{region '#Template'}
	{attribute 'Version' := '5.0.0.0'}
	{attribute 'Tags' := '"LCID": "1031", "Text": "Gebäudeautomation, Wetterdaten"'}
	{attribute 'Tags' := '"LCID": "1033", "Text": "Building automation, Weather data"'}
	{attribute 'Using' := '"Type": "Template", "URI": "BA2_Param"'}
	{attribute 'Using' := '"Type": "Template", "URI": "Site"'}		  
	{attribute 'Using' := '"Type": "Template", "URI": "ST_BA_GeneralSettings"'}
	{attribute 'Description' := '"LCID": "1031", "Text": "Gebäude Wetterdaten"'}
	{attribute 'Description' := '"LCID": "1033", "Text": "Building Weather data"'}
{endregion}
FUNCTION_BLOCK FB_BA_WeatherData EXTENDS FB_BA_View
VAR_INPUT CONSTANT
	WthParam				: FB_BA_WeatherParameter;	
END_VAR
VAR // added by the converter: edge detectors and wires of the graphical bodies
    _s1 : ST_BA_GeneralSettings;
END_VAR

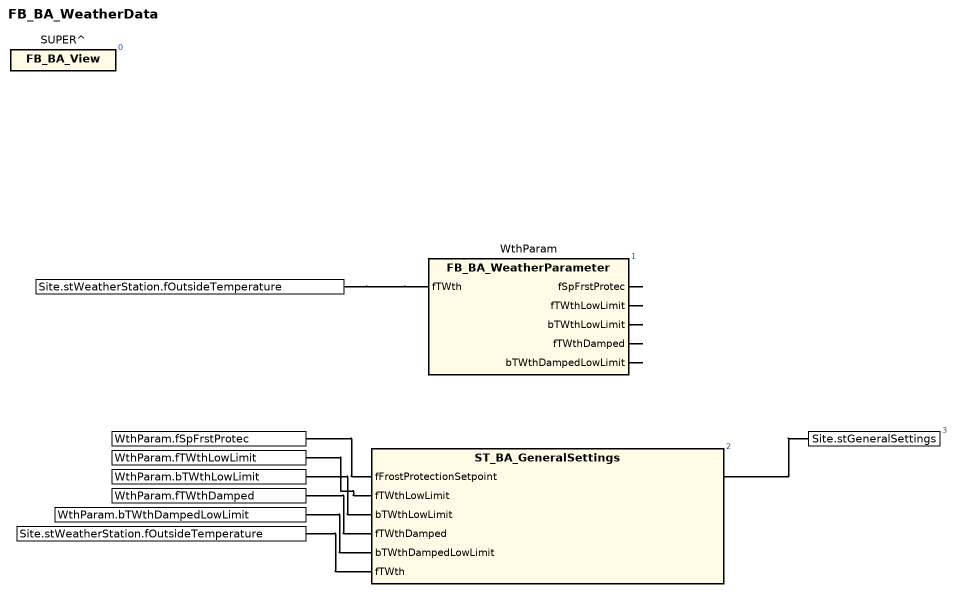
SUPER^(); // FB_BA_View
WthParam(fTWth := Site.stWeatherStation.fOutsideTemperature); // FB_BA_WeatherParameter
// compose _s1 : ST_BA_GeneralSettings
_s1.fFrostProtectionSetpoint := WthParam.fSpFrstProtec;
_s1.fTWthLowLimit := WthParam.fTWthLowLimit;
_s1.bTWthLowLimit := WthParam.bTWthLowLimit;
_s1.fTWthDamped := WthParam.fTWthDamped;
_s1.bTWthDampedLowLimit := WthParam.bTWthDampedLowLimit;
_s1.fTWth := Site.stWeatherStation.fOutsideTemperature;
Site.stGeneralSettings := _s1;

METHOD FB_init : BOOL
VAR_INPUT
	bInitRetains : BOOL; // if TRUE, the retain variables are initialized (warm start / cold start)
	bInCopyCode : BOOL;  // if TRUE, the instance afterwards gets moved into the copy code (online change)
END_VAR
WthParam.iParent			:= THIS^;
WthParam.iLabel				:= LblCtl_WeatherParameters;
WthParam.eDPADMode			:= E_BA_DPADMode.eInclude;
END_METHOD

END_FUNCTION_BLOCK

(* stored: Version 1.1.0.1, ProductVersion 3.1.4024.12
   POU FB_BA_WeatherData: Id {e624f4a8-3ee8-4303-89cf-7d8ec91ad3de}, SpecialFunc None
   Method FB_init: Id {62861317-b611-4c3c-a458-a471ea9188ab} *)
